# EPICS substitutions: Ophir5087.substitutions
file Ophir5087.template {
pattern {P, PORT}
    {"BL4A:SF:OPHIR1", "OP1"}
    {"BL4A:SF:OPHIR2", "OP2"}

}
